(* IEC 61131-3 sources: RL_MAR/experiments/comparison/llm4plc/results/Qwen-Qwen3.5-9B_20260506_150728/20260506_165016, 4 files *)

(* ---- generated_code_iteration_0.st ---- *)
START_ST
FUNCTION_BLOCK SandwichMaker
VAR_INPUT
    BreadFeeder : BOOL; (* Input: Detects the presence of bread slices *)
    Ingredient1 : BOOL; (* Input: Detects the presence of Ingredient 1 (e.g., cheese) *)
    Ingredient2 : BOOL; (* Input: Detects the presence of Ingredient 2 (e.g., lettuce) *)
    Ingredient3 : BOOL; (* Input: Detects the presence of Ingredient 3 (e.g., tomatoes) *)
    Condiment1 : BOOL; (* Input: Detects the presence of Condiment 1 (e.g., mayo) *)
    Condiment2 : BOOL; (* Input: Detects the presence of Condiment 2 (e.g., mustard) *)
END_VAR
VAR_OUTPUT
    ConveyorMotor : BOOL; (* Output: Controls the conveyor belt motor *)
    AssembleMotor : BOOL; (* Output: Controls the sandwich assembly motor *)
END_VAR
VAR
    SliceCount : INT := 0; (* Counter for bread slices *)
    State : INT := 0; (* Current State: 0=IDLE, 1=CONVEYING, 2=ASSEMBLING *)
    AllIngredientsPresent : BOOL; (* Helper variable for ingredient check *)
END_VAR
END_VAR

BEGIN
    (* 1. Determine if all ingredients and condiments are present *)
    AllIngredientsPresent := (Ingredient1 AND Ingredient2 AND Ingredient3 AND Condiment1 AND Condiment2);

    (* 2. State Machine Logic *)
    CASE State OF
        (* STATE 0: IDLE *)
        (* Description: System is waiting for bread. Both motors are OFF. *)
        0 ->
            ConveyorMotor := FALSE;
            AssembleMotor := FALSE;

            (* Transition to STATE 1 (CONVEYING) *)
            (* Condition: Bread is detected *)
            IF BreadFeeder THEN
                State := 1;
            END_IF;

        (* STATE 1: CONVEYING *)
        (* Description: Bread has been detected. ConveyorMotor is ON. SliceCount is incremented. *)
        1 ->
            ConveyorMotor := TRUE;
            AssembleMotor := FALSE;

            (* Increment slice count if bread is present *)
            IF BreadFeeder THEN
                SliceCount := SliceCount + 1;
            END_IF;

            (* Check transition conditions *)
            (* Transition to STATE 2 (ASSEMBLING): Count >= 2 AND All Ingredients Present *)
            IF (SliceCount >= 2) AND AllIngredientsPresent THEN
                State := 2;
            (* Transition to STATE 0 (IDLE/RESET): Bread leaves sensor (BreadFeeder becomes FALSE) *)
            (* This implies the sandwich has moved past the sensor, so we reset for the next cycle *)
            ELSEIF NOT BreadFeeder THEN
                State := 0;
                SliceCount := 0; (* Reset counter when bread is no longer detected *)
            END_IF;

        (* STATE 2: ASSEMBLING *)
        (* Description: At least two bread slices are present AND all ingredients/condiments are present. *)
        (* AssembleMotor is ON. ConveyorMotor remains ON to push the sandwich. *)
        2 ->
            ConveyorMotor := TRUE;
            AssembleMotor := TRUE;

            (* Logic to exit State 2 *)
            (* Transition to STATE 0 (RESET): Bread leaves sensor (BreadFeeder becomes FALSE) *)
            (* This signifies the sandwich is complete and leaving the station *)
            IF NOT BreadFeeder THEN
                State := 0;
                SliceCount := 0; (* Reset counter *)
            (* Transition back to STATE 1 (CONVEYING): If bread is present but conditions fail *)
            (* e.g., Count < 2 or Ingredients missing *)
            ELSEIF NOT ((SliceCount >= 2) AND AllIngredientsPresent) THEN
                State := 1;
            END_IF;

        (* STATE 3: RESET (Not explicitly used in the simplified flow above as transitions go 2->0 directly,
           but included here for completeness if logic were expanded. Based on plan, 0 covers IDLE/RESET. *)
        3 ->
            ConveyorMotor := FALSE;
            AssembleMotor := FALSE;
            SliceCount := 0;
    ENDCASE
END_FUNCTION_BLOCK
END_ST

(* ---- generated_code_iteration_1.st ---- *)
START_REASON
The error "发现非预期的记号'END_VAR'" (Unexpected token 'END_VAR') occurs because the variable section for the FUNCTION_BLOCK was closed prematurely. In IEC 61131-3 Structured Text, the `END_VAR` keyword must appear only once at the very end of the variable declaration block, immediately before the `BEGIN` keyword that starts the executable logic.

In the provided code, there was an extra `END_VAR` placed after the `VAR` section (closing the inputs/outputs/variables) but before the `BEGIN` statement. This caused the compiler to expect the start of the program logic (`BEGIN`) instead of finding another variable terminator.

The fix involves removing the erroneous `END_VAR` between the `VAR` section and the `BEGIN` statement, ensuring the structure follows:
1. `FUNCTION_BLOCK Name`
2. `VAR_INPUT ... END_VAR` (Optional if inputs are mixed, but usually `VAR_INPUT` ends with `END_VAR` only if followed by `VAR_OUTPUT` or `VAR` in a specific way, OR simply grouping them under one `VAR` block).
   *Correction on IEC 61131-3 Syntax*: Actually, the standard syntax allows:
   `VAR_INPUT ... END_VAR`
   `VAR_OUTPUT ... END_VAR`
   `VAR ... END_VAR`
   OR
   `VAR_INPUT ... VAR_OUTPUT ... VAR ... END_VAR` (Single block).

Looking at the original code:
```
VAR_INPUT ... END_VAR
VAR_OUTPUT ... END_VAR
VAR ... END_VAR
END_VAR  <-- This is the duplicate causing the error.
BEGIN
```
The code had three separate variable blocks (Input, Output, Var) which is valid, but then it had a fourth `END_VAR` floating before `BEGIN`. This is the syntax error. I will consolidate the variable declarations into a single `VAR` block or ensure the `END_VAR` count matches the `VAR`/`VAR_INPUT`/`VAR_OUTPUT` start tags correctly. The most robust fix for this specific error is to remove the stray `END_VAR` before `BEGIN`.

Wait, looking closer at the provided code:
```
VAR_INPUT
    ...
END_VAR
VAR_OUTPUT
    ...
END_VAR
VAR
    ...
END_VAR
END_VAR  <-- This line is the problem.
BEGIN
```
The code has `VAR_INPUT`...`END_VAR`, `VAR_OUTPUT`...`END_VAR`, `VAR`...`END_VAR`. That is three blocks. Then there is a fourth `END_VAR`. This is definitely the issue. I will remove the extra `END_VAR` and ensure the structure is clean.

Also, I need to make sure I don't change the logic, just the syntax.

START_ST
FUNCTION_BLOCK SandwichMaker
VAR_INPUT
    BreadFeeder : BOOL;
    Ingredient1 : BOOL;
    Ingredient2 : BOOL;
    Ingredient3 : BOOL;
    Condiment1 : BOOL;
    Condiment2 : BOOL;
END_VAR
VAR_OUTPUT
    ConveyorMotor : BOOL;
    AssembleMotor : BOOL;
END_VAR
VAR
    SliceCount : INT := 0;
    State : INT := 0;
    AllIngredientsPresent : BOOL;
END_VAR
BEGIN
    (* 1. Determine if all ingredients and condiments are present *)
    AllIngredientsPresent := (Ingredient1 AND Ingredient2 AND Ingredient3 AND Condiment1 AND Condiment2);

    (* 2. State Machine Logic *)
    CASE State OF
        (* STATE 0: IDLE *)
        0 ->
            ConveyorMotor := FALSE;
            AssembleMotor := FALSE;

            (* Transition to STATE 1 (CONVEYING) *)
            IF BreadFeeder THEN
                State := 1;
            END_IF;

        (* STATE 1: CONVEYING *)
        1 ->
            ConveyorMotor := TRUE;
            AssembleMotor := FALSE;

            (* Increment slice count if bread is present *)
            IF BreadFeeder THEN
                SliceCount := SliceCount + 1;
            END_IF;

            (* Check transition conditions *)
            IF (SliceCount >= 2) AND AllIngredientsPresent THEN
                State := 2;
            ELSEIF NOT BreadFeeder THEN
                State := 0;
                SliceCount := 0;
            END_IF;

        (* STATE 2: ASSEMBLING *)
        2 ->
            ConveyorMotor := TRUE;
            AssembleMotor := TRUE;

            (* Logic to exit State 2 *)
            IF NOT BreadFeeder THEN
                State := 0;
                SliceCount := 0;
            ELSEIF NOT ((SliceCount >= 2) AND AllIngredientsPresent) THEN
                State := 1;
            END_IF;

        (* STATE 3: RESET (Unused in current flow but defined for completeness) *)
        3 ->
            ConveyorMotor := FALSE;
            AssembleMotor := FALSE;
            SliceCount := 0;
    ENDCASE
END_FUNCTION_BLOCK
END_ST
END_REASON

(* ---- generated_code_iteration_2.st ---- *)
START_REASON
The previous code failed validation due to an encoding issue where the Chinese comment characters `(*` and `*)` were likely interpreted or encoded incorrectly (specifically the byte `0xa2` corresponds to a full-width or special character in GBK encoding, often appearing when Chinese punctuation is used in a context expecting ASCII or UTF-8). The compiler (ANTLR/CODESYS) cannot parse these characters.

To fix this:
1.  Replace all Chinese comments with standard English comments.
2.  Ensure the Structured Text syntax strictly follows IEC 61131-3 standards.
3.  Maintain the `FUNCTION_BLOCK` structure with correct `VAR_INPUT`, `VAR_OUTPUT`, `VAR`, and `END_VAR` placements.
4.  Remove any stray `END_VAR` tokens that might have been part of the previous erroneous structure.

The logic remains: A state machine controlling a sandwich maker based on ingredient presence and bread feeding.
START_ST
FUNCTION_BLOCK SandwichMaker
VAR_INPUT
    BreadFeeder : BOOL;
    Ingredient1 : BOOL;
    Ingredient2 : BOOL;
    Ingredient3 : BOOL;
    Condiment1 : BOOL;
    Condiment2 : BOOL;
END_VAR
VAR_OUTPUT
    ConveyorMotor : BOOL;
    AssembleMotor : BOOL;
END_VAR
VAR
    SliceCount : INT := 0;
    State : INT := 0;
    AllIngredientsPresent : BOOL;
END_VAR
BEGIN
    (* Determine if all ingredients and condiments are present *)
    AllIngredientsPresent := (Ingredient1 AND Ingredient2 AND Ingredient3 AND Condiment1 AND Condiment2);

    (* State Machine Logic *)
    CASE State OF
        (* STATE 0: IDLE *)
        0 ->
            ConveyorMotor := FALSE;
            AssembleMotor := FALSE;

            (* Transition to STATE 1 (CONVEYING) *)
            IF BreadFeeder THEN
                State := 1;
            END_IF;

        (* STATE 1: CONVEYING *)
        1 ->
            ConveyorMotor := TRUE;
            AssembleMotor := FALSE;

            (* Increment slice count if bread is present *)
            IF BreadFeeder THEN
                SliceCount := SliceCount + 1;
            END_IF;

            (* Check transition conditions *)
            IF (SliceCount >= 2) AND AllIngredientsPresent THEN
                State := 2;
            ELSEIF NOT BreadFeeder THEN
                State := 0;
                SliceCount := 0;
            END_IF;

        (* STATE 2: ASSEMBLING *)
        2 ->
            ConveyorMotor := TRUE;
            AssembleMotor := TRUE;

            (* Logic to exit State 2 *)
            IF NOT BreadFeeder THEN
                State := 0;
                SliceCount := 0;
            ELSEIF NOT ((SliceCount >= 2) AND AllIngredientsPresent) THEN
                State := 1;
            END_IF;

        (* STATE 3: RESET (Unused in current flow but defined for completeness) *)
        3 ->
            ConveyorMotor := FALSE;
            AssembleMotor := FALSE;
            SliceCount := 0;
    ENDCASE
END_FUNCTION_BLOCK
END_ST
END_REASON

(* ---- generated_code_iteration_3.st ---- *)
START_REASON
The previous code failed CODESYS validation with the error: "应该用';' 替换'AllIngredientsPresent'" (Should replace 'AllIngredientsPresent' with ';').

This error occurs because in IEC 61131-3 Structured Text, every executable statement must end with a semicolon (`;`). The line:
`AllIngredientsPresent := (Ingredient1 AND Ingredient2 AND Ingredient3 AND Condiment1 AND Condiment2);`
was likely missing the semicolon in the previous iteration or the parser is strict about line endings. Although the provided code block in the prompt *shows* a semicolon, the specific error message from the toolchain implies that the actual generated output lacked it or the line was treated as incomplete.

Additionally, while the logic is sound, I will ensure strict adherence to IEC 61131-3 standards:
1.  Ensure every assignment and control structure statement ends with `;`.
2.  Keep comments in English (`(* ... *)`) to avoid encoding issues.
3.  Maintain the `FUNCTION_BLOCK` structure.
4.  Ensure `END_VAR` is used correctly to close variable sections.

The fix involves explicitly ensuring the assignment of `AllIngredientsPresent` is terminated with a semicolon and verifying all other statements follow suit.
END_REASON
START_ST
FUNCTION_BLOCK SandwichMaker
VAR_INPUT
    BreadFeeder : BOOL;
    Ingredient1 : BOOL;
    Ingredient2 : BOOL;
    Ingredient3 : BOOL;
    Condiment1 : BOOL;
    Condiment2 : BOOL;
END_VAR
VAR_OUTPUT
    ConveyorMotor : BOOL;
    AssembleMotor : BOOL;
END_VAR
VAR
    SliceCount : INT := 0;
    State : INT := 0;
    AllIngredientsPresent : BOOL;
END_VAR
BEGIN
    (* Determine if all ingredients and condiments are present *)
    AllIngredientsPresent := (Ingredient1 AND Ingredient2 AND Ingredient3 AND Condiment1 AND Condiment2);

    (* State Machine Logic *)
    CASE State OF
        (* STATE 0: IDLE *)
        0 ->
            ConveyorMotor := FALSE;
            AssembleMotor := FALSE;

            (* Transition to STATE 1 (CONVEYING) *)
            IF BreadFeeder THEN
                State := 1;
            END_IF;

        (* STATE 1: CONVEYING *)
        1 ->
            ConveyorMotor := TRUE;
            AssembleMotor := FALSE;

            (* Increment slice count if bread is present *)
            IF BreadFeeder THEN
                SliceCount := SliceCount + 1;
            END_IF;

            (* Check transition conditions *)
            IF (SliceCount >= 2) AND AllIngredientsPresent THEN
                State := 2;
            ELSEIF NOT BreadFeeder THEN
                State := 0;
                SliceCount := 0;
            END_IF;

        (* STATE 2: ASSEMBLING *)
        2 ->
            ConveyorMotor := TRUE;
            AssembleMotor := TRUE;

            (* Logic to exit State 2 *)
            IF NOT BreadFeeder THEN
                State := 0;
                SliceCount := 0;
            ELSEIF NOT ((SliceCount >= 2) AND AllIngredientsPresent) THEN
                State := 1;
            END_IF;

        (* STATE 3: RESET (Unused in current flow but defined for completeness) *)
        3 ->
            ConveyorMotor := FALSE;
            AssembleMotor := FALSE;
            SliceCount := 0;
    ENDCASE
END_FUNCTION_BLOCK
END_ST
END_REASON
